FUNCTION_BLOCK FB_Reaktoreinheit IMPLEMENTS I_Reaktor
VAR_INPUT
	I_SW				:SystemStatusWord;			// Reaktorrückmeldung von OPC UA Schnittstelle
	I_Parameter			:SystemControlWord; 		// Prozessparameter 
END_VAR
	
VAR_OUTPUT
	O_CW			:SystemControlWord; 		// Prozessparameter für OPC UA Schnittstelle
END_VAR

VAR
	V_Status		:INT;						// Variable für internes handling der Eigenschaft
END_VAR

// Setzen der internen Variablen
V_Status := P_Status;

METHOD M_A_OFF : BOOL
VAR_INPUT
END_VAR
O_CW.PowerOn := FALSE;
END_METHOD

METHOD M_A_ON : BOOL
VAR_INPUT
END_VAR
O_CW.PowerOn := TRUE;
END_METHOD

METHOD M_A_START : BOOL
VAR_INPUT
END_VAR
O_CW := I_Parameter;
END_METHOD

METHOD M_A_STOP : BOOL
VAR_INPUT
END_VAR
O_CW.SekReakt := 0;
O_CW.Leitung := 0;
O_CW.Temp := 0;
O_CW.Enlteermenge := 0;
O_CW.Pumpmenge := 0;
O_CW.Haltedauer := T#0S;
O_CW.Ruehrdauer := T#0S;
O_CW.Wartedauer := T#0S;
O_CW.Zirkulierdauer := T#0S;
END_METHOD

METHOD M_M_OFF : BOOL
VAR_INPUT
END_VAR
O_CW.PowerOn := FALSE;
END_METHOD

METHOD M_M_ON : BOOL
VAR_INPUT
END_VAR
O_CW.PowerOn := TRUE;
END_METHOD

METHOD M_M_START : BOOL
VAR_INPUT
END_VAR
O_CW := I_Parameter;
END_METHOD

METHOD M_M_STOP : BOOL
VAR_INPUT
END_VAR
O_CW.SekReakt := 0;
O_CW.Leitung := 0;
O_CW.Temp := 0;
O_CW.Enlteermenge := 0;
O_CW.Pumpmenge := 0;
O_CW.Haltedauer := T#0S;
O_CW.Ruehrdauer := T#0S;
O_CW.Wartedauer := T#0S;
O_CW.Zirkulierdauer := T#0S;
END_METHOD

PROPERTY P_Status : INT
GET
IF I_SW.PrimReady THEN
	P_Status := 1;
END_IF

IF I_SW.PrimActiv THEN
	P_Status := 2;
END_IF
END_GET
END_PROPERTY

END_FUNCTION_BLOCK

(* stored: Version 1.1.0.1, ProductVersion 3.1.4024.12
   POU FB_Reaktoreinheit: Id {e70a7bfb-3a77-4ac5-848e-915860a164c8}, SpecialFunc None
   Method M_A_OFF: Id {b86c77af-8803-46fa-8eaa-5ebfd1812af6}
   Method M_A_ON: Id {ce3ee9e0-881b-473a-80ba-d0fc2959046e}
   Method M_A_START: Id {465c5990-02eb-4d01-a0be-c08f377138c6}
   Method M_A_STOP: Id {d8444895-e01a-478c-8eaf-23650e449549}
   Method M_M_OFF: Id {15ab24aa-7a53-42fc-8b32-af1250aef26d}
   Method M_M_ON: Id {2cc463e2-7a73-4f79-8ecd-c91093a26e4b}
   Method M_M_START: Id {712c9664-1124-4804-9d76-723ce000bf52}
   Method M_M_STOP: Id {45bf1e14-c8df-4553-b479-f9eed412350d}
   Property P_Status: Id {23579e58-21f7-4d5c-8cdd-0dc574eac682}
   Get Get: Id {36f9b8e6-75d2-4ae3-a343-599d77dd5e02} *)
